Staubli VAL3: onEnterEvent.pgx

program onEnterEvent(string x_sName)
  local num l_nSize[4]
  local num i
  local string l_sProg
  local num l_nIndex
  local num l_nPosition[4]
  local string l_sEmpty
begin
  //
  // NB sEvent is the selected
  // element in the LIST
  //
  call pallet:getPalletPos(x_sName,l_nPosition)
  call pallet:getSizePallet(x_sName,l_nSize)
  //
  if nIndex>=0
    i=find(sEvent,">")+1
  endIf
  //
  // clean the line
  call use:listcursor(use:nView,false)
  //
  if l_nSize>1
    // absolute
    l_sEmpty=""
    l_nPosition=l_nPosition+1
    call use:changeValue(l_nPosition,1,l_nSize,i+40-use:nBottomX,use:nView+1,l_sEmpty)
    call pallet:setPalletPos(x_sName,l_nPosition-1)
    // refresh it
    call buildList()
  endIf
  use:bUseRefresh=true
end
